TYPE TestStruct :
STRUCT
	i: INT;
	b: REAL;
	test_array_st: ARRAY[0..12] OF LREAL;
END_STRUCT
END_TYPE

(* stored: Version 1.1.0.1
   DUT TestStruct: Id {ebcb16e4-fd99-4454-afea-c9751729e78f} *)
